// TwinCAT 3 PLC project _2_4_Timer_TON
// ProgramVersion: 3.1.4020.2
// libraries:
//   Tc2_Standard, * (Beckhoff Automation GmbH)
//   Tc2_System, * (Beckhoff Automation GmbH)
//   Tc3_Module, * (Beckhoff Automation GmbH)
// project tree:
//   / GlobalTextList.TcGTLO, PlcTask.TcTTO, Visualization Manager.TcVMO (not stored)
//   POUs/ MAIN.TcPOU
//   VISUs/ Visualization.TcVIS
// (motion and I/O tree: see PLC project 1calcul)
// real-time tasks:
//   TASK PlcTask: cycle T#1ms, priority 20, ADS port 350
// variable links:

CONFIGURATION _2_4_Timer_TON
    RESOURCE PLC ON TwinCAT3
        TASK PlcTask(INTERVAL := T#1ms, PRIORITY := 20);
        PROGRAM MAIN WITH PlcTask : MAIN;
    END_RESOURCE
END_CONFIGURATION

// ---- POUs/MAIN.TcPOU
PROGRAM MAIN
VAR
	MxEnableTimer:BOOL :=TRUE;
	MxLight: BOOL :=FALSE;
	MxTimeDone: BOOL := FALSE;
	Timer: TON;
	MxOn: BOOL:=FALSE;
END_VAR

//Timer
Timer(IN:=MxEnableTimer , PT:=T#1000MS , Q=> , ET=> );


//actions to take to reset Timer and change LightStatus
IF Timer.Q THEN
		MxLight:=NOT MxLight;
		MxEnableTimer:=FALSE;
	ELSIF MxOn AND NOT MxEnableTimer THEN
			MxEnableTimer:= TRUE;
END_IF

END_PROGRAM

// ---- VISUs/Visualization.TcVIS
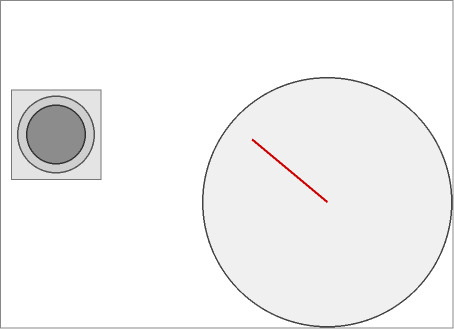
VISUALIZATION Visualization  // 454x329
    PushSwitchLed (11,64 90x141), variable: .MAIN.MxOn, behaviour: TOGGLE, style: Switch-PushSwitchLed-Gray
    Meter180 (202,77 250x250), style: Meter-Meter180-Gray, scale format: %.1f, scale 0..1000
END_VISUALIZATION
